FUNCTION_BLOCK ASSEMBLE_AD_FROM_AB (* this Function combines the 4 AB (BYTE) adapters to a AD (DWORD) *)
  (* Standard: 61499-2; Description: Copyright (c) 2026 Meisterschulen am Ostbahnhof SPDX-License-Identifier: EPL-2.0 *)
  (* Version 1.0, 2026-05-16, Franz Höpfinger, Meisterschulen am Ostbahnhof, initial API and implementation and/or initial documentation *)
  PACKAGE adapter::assembling;
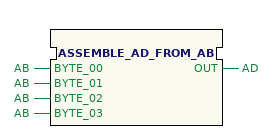
  SOCKETS
    BYTE_00 : adapter::types::unidirectional::AB; (* Byte 0 *)
    BYTE_01 : adapter::types::unidirectional::AB; (* Byte 1 *)
    BYTE_02 : adapter::types::unidirectional::AB; (* Byte 2 *)
    BYTE_03 : adapter::types::unidirectional::AB; (* Byte 3 *)
  END_SOCKETS
  PLUGS
    OUT : adapter::types::unidirectional::AD; (* DWORD Output *)
  END_PLUGS
END_FUNCTION_BLOCK
